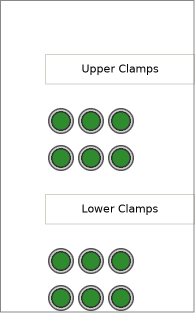
VISUALIZATION Visualization  // 195x313
    Lamp1 (46,106 30x30), variable: MAIN.simClampUpper.I_bCmdValveOff, style: Lamp-Lamp1-Green
    Textfield (45,54 150x30), "Upper Clamps"
    Lamp1 (46,143 30x30), variable: MAIN.simClampUpper.I_bCmdValveOn, style: Lamp-Lamp1-Green
    Lamp1 (76,143 30x30), variable: MAIN.simClampUpper.Q_bStaFeedbackOn, style: Lamp-Lamp1-Green
    Lamp1 (76,106 30x30), variable: MAIN.simClampUpper.Q_bStaFeedbackOff, style: Lamp-Lamp1-Green
    Lamp1 (106,106 30x30), variable: MAIN.simClampUpper.Q_bStaFeedbackOff2, style: Lamp-Lamp1-Green
    Lamp1 (106,143 30x30), variable: MAIN.simClampUpper.Q_bStaFeedbackOn2, style: Lamp-Lamp1-Green
    Lamp1 (46,246 30x30), variable: MAIN.simClampLower.I_bCmdValveOff, style: Lamp-Lamp1-Green
    Textfield (45,194 150x30), "Lower Clamps"
    Lamp1 (46,283 30x30), variable: MAIN.simClampLower.I_bCmdValveOn, style: Lamp-Lamp1-Green
    Lamp1 (76,283 30x30), variable: MAIN.simClampLower.Q_bStaFeedbackOn, style: Lamp-Lamp1-Green
    Lamp1 (76,246 30x30), variable: MAIN.simClampLower.Q_bStaFeedbackOff, style: Lamp-Lamp1-Green
    Lamp1 (106,246 30x30), variable: MAIN.simClampLower.Q_bStaFeedbackOff2, style: Lamp-Lamp1-Green
    Lamp1 (106,283 30x30), variable: MAIN.simClampLower.Q_bStaFeedbackOn2, style: Lamp-Lamp1-Green
END_VISUALIZATION

(* stored: Version 1.1.0.1, ProductVersion 3.1.4024.12
   Visu Visualization: Id {f5e16759-9129-4da3-9ed9-47cf081874d4} *)
